TYPE commUnitConfig :
STRUCT
	unitId : WORD; //0
	configId: WORD;//1
	value : DWORD;//2
END_STRUCT
END_TYPE

(* stored: Version 1.1.0.1, ProductVersion 3.1.4022.10
   DUT commUnitConfig: Id {4b0a5ad5-bbdc-45ab-a479-8df6412da007} *)
